Fanuc KAREL source: kt00370.KL

-- PROVISIONAL review KL for V770-1; original PC SHA256 fbc4f66bb2fb914f8d781b48be60f73ba6c1a8bcfc0fb51cf221ae649475bdfe
-- Incomplete behavior may be omitted. Consult companion uncertainty JSON. Do not deploy.
PROGRAM KT00370
%NOLOCKGROUP
VAR
  R1 : REAL
  R2 : REAL
  OUT : BOOLEAN
BEGIN
  -- UNRESOLVED_PC offsets 5-16; opcodes 2E,23
  -- UNRESOLVED_PC offsets 21-32; opcodes 2E,23
  -- UNRESOLVED_PC offsets 37-48; opcodes 2E,23
  -- UNRESOLVED_PC offsets 53-64; opcodes 2E,23
  -- UNRESOLVED_PC offsets 69-88; opcodes 21,21,70,23
  -- UNRESOLVED_PC offsets 93-97; opcodes 7F
END KT00370
